TYPE ST_PCMSystemSetParameters :
STRUCT
	nControlModeAlgorithm : E_PCMSystemControlMode;
	nControlModeManual : E_PCMSystemControlMode;
END_STRUCT
END_TYPE

(* stored: Version 1.1.0.1, ProductVersion 3.1.4024.10
   DUT ST_PCMSystemSetParameters: Id {2bfe854b-bd7a-43e8-a6f6-8d605b1dc106} *)
